FUNCTION_BLOCK AxisPower EXTENDS TaskBase
VAR
	mcPower : Tc2_MC2.MC_Power;
	AxisReference : REFERENCE TO Tc2_MC2.AXIS_REF;
	EnableAxis : BOOL;
END_VAR

METHOD Abort : BOOL
mcPower.Enable := mcPower.Enable_Negative := mcPower.Enable_Positive := FALSE;
_busy := FALSE;
EnableAxis := FALSE;
Abort := TRUE;
State := 0;
END_METHOD

PROPERTY Busy : BOOL
GET
Busy := _busy;
END_GET
END_PROPERTY

METHOD Cycle : BOOL
VAR_INPUT
END_VAR
CASE State OF
	0:
		IF EnableAxis THEN
			_done := FALSE;
			_error := FALSE;
			_busy := TRUE;
			mcPower.Enable := mcPower.Enable_Negative := mcPower.Enable_Positive := TRUE;
			mcPower.Override := 100;
			State := 10;
		END_IF
	
	10:
		IF mcPower.Status THEN
			_busy := FALSE;
			_done := TRUE;
			state := 20;
		END_IF
	
	20:
		IF NOT EnableAxis THEN
			_done := FALSE;
			_busy := TRUE;
			mcPower.Enable := mcPower.Enable_Negative := mcPower.Enable_Positive := FALSE;
			State := 30;
		END_IF
	30:
		IF NOT mcPower.Status THEN
			_busy := FALSE;
			_done := TRUE;
			state := 0;
		END_IF
END_CASE

mcPower(Axis := AxisReference);
END_METHOD

METHOD Disable : BOOL
VAR_INPUT
END_VAR
IF NOT EnableAxis THEN
	RETURN;
END_IF
Disable := TRUE;
EnableAxis := FALSE;
END_METHOD

PROPERTY Done : BOOL
GET
Done := _done;
END_GET
END_PROPERTY

METHOD Enable : BOOL
VAR_INPUT
END_VAR
IF EnableAxis THEN
	RETURN;
END_IF
Enable := EnableAxis := true;
END_METHOD


PROPERTY Error : BOOL
GET
Error := _error;
END_GET
END_PROPERTY

METHOD FB_init : BOOL
VAR_INPUT
	bInitRetains : BOOL; // if TRUE, the retain variables are initialized (warm start / cold start)
	bInCopyCode : BOOL;  // if TRUE, the instance afterwards gets moved into the copy code (online change)
	axis : reference TO AXIS_REF;
END_VAR
AxisReference REF= axis;
END_METHOD

END_FUNCTION_BLOCK

(* stored: Version 1.1.0.1, ProductVersion 3.1.4024.12
   POU AxisPower: Id {cf8d7780-536f-48f2-8eb4-f2d08824929f}, SpecialFunc None
   Method Abort: Id {6b214ba9-44b4-4668-9ec2-8eddbec189ec}
   Property Busy: Id {ef0f4437-de71-4221-a0af-37624a426c16}
   Get Get: Id {811a31bb-e198-434f-898d-917e03bf6183}
   Method Cycle: Id {49735321-892e-4ec1-aa25-952ce1fe7601}
   Method Disable: Id {71e12fcb-ea2b-4a80-97e6-c20b6299e2da}
   Property Done: Id {3edec79a-21aa-4354-b705-f4ba8d01278c}
   Get Get: Id {0fac9851-7ef7-47cb-bfc6-71b8d612bcb6}
   Method Enable: Id {a6939086-c52d-4f49-9683-237a63574b37}
   Property Error: Id {8a127411-a21f-4341-9085-d8abfe79a613}
   Get Get: Id {63932449-f083-4a78-aad0-5b7fc0222e68}
   Method FB_init: Id {4f3f0882-eaae-4802-8592-bb1a398d403a} *)
